TYPE EtcSlaveBase_82538BE2 :
STRUCT
END_STRUCT
END_TYPE

(* stored: Version 1.2.0.0, ProductVersion 3.1.4024.9
   DUT EtcSlaveBase_82538BE2: Id {7ef2583b-7db4-44f4-8e3d-fd2c5b9a8572} *)
